FUNCTION_BLOCK FB_PersistentDataStorage_TestDouble IMPLEMENTS I_PersistentDataStorage
VAR
END_VAR

{warning 'Add property implementation'}
PROPERTY TriggerWriteOfPersistentData : BOOL
GET
END_GET
SET
END_SET
END_PROPERTY

END_FUNCTION_BLOCK

(* stored: Version 1.1.0.1
   POU FB_PersistentDataStorage_TestDouble: Id {44bca275-b094-4c6c-b0de-84278cf52d1a}, SpecialFunc None
   Property TriggerWriteOfPersistentData: Id {236bb73c-de8d-49a9-bedf-b9e640dcf1eb}
   Get Get: Id {afbc1d73-9208-4dff-a219-f99087ac23a8}
   Set Set: Id {2377f624-d6a9-4b8b-8794-540331f45295} *)
